Staubli VAL3: find.pgx

public program find(string& x_sItem[] (dimensions=1), bool& x_bFound[] (dimensions=1))
  local num i
  local num l_nSize
  local string l_sEvent
begin
  // check if the item has been found
  x_bFound=isDefined(saveProg:pProg[x_sItem])
end
